FUNCTION_BLOCK FB_MyFB1
VAR_INPUT
END_VAR
VAR_OUTPUT
END_VAR
VAR
END_VAR

END_FUNCTION_BLOCK

(* stored: Version 1.1.0.1, ProductVersion 3.1.4024.14
   POU FB_MyFB1: Id {54c242be-e4cc-440c-9fd7-442f5d1fb5a7}, SpecialFunc None *)
